{attribute 'object_name' := 'sta_EOFFBusy'}
METHOD sta_EOFFBusy : BOOL
                        // state implemetation
//--------------------------------------------------------------------------------------
// Entry action
	IF (me.StateMachine.intState<>me.StateMachine.intStateLastCycle) THEN
		me.StateMachine.intStateLastCycle := me.StateMachine.intState;
	END_IF

	
//--------------------------------------------------------------------------------------
// Cyclic action
	IF (me.StateMachine.intState=me.StateMachine.intStateLastCycle) THEN
		
		// In case of an emergency, set all childs to off 
		// Set in cyclic action because of possible errors or manual/auto changes!
		SUPER^.SetAllChildCmd(BASE_PLC.cCMD_OFF);

		// check if all childs have reached the state
		IF CheckAllChildState(cSTA_OFF) THEN
			me.StateMachine.intStateNext := cSTA_EOFF;
		END_IF
	END_IF

	
//--------------------------------------------------------------------------------------
// Exit action
	IF (me.StateMachine.intState<>me.StateMachine.intStateNext) THEN
		;
	END_IF
                      
END_METHOD

{attribute 'object_name' := 'sta_STOP'}
METHOD sta_STOP : BOOL
                        // state implemetation
//--------------------------------------------------------------------------------------
// Entry action
	IF (me.StateMachine.intState<>me.StateMachine.intStateLastCycle) THEN
		me.StateMachine.intStateLastCycle := me.StateMachine.intState;
	END_IF


//--------------------------------------------------------------------------------------
// Cyclic action
	IF (me.StateMachine.intState=me.StateMachine.intStateLastCycle) THEN
		
		// State Change Condition
		IF (me.Alarm.eActivAlmClass<E_AlmClass.TSTOP) THEN
			IF (me.intCmd=cCMD_RUN) THEN
				IF (SIf_In^.bolReady.intern OR SIf_Cfg^.bolIgnoreReadyInput) THEN 
					me.StateMachine.intStateNext := cSTA_RUNBusy;
				ELSE
					//SIf_MOD.Alm[E_ALM_MOD.NextModuleNotReadyWarning].strText := 'Next Module is not Ready';
					pfbAlarmCtrl^.setAlarm(CIf.Info.intCtrlId,E_ALM_MOD.NextModuleNotReadyWarning,0,ADR(SIf_MOD.Alm),E_AlmState.RST,CIf.Job.eMe_ActivAlmClass);
					CIf.Job.intACmd := cCMD_DONE;
				END_IF
			ELSIF (me.intCmd=cCMD_STANDBY) THEN
				IF (SIf_In^.bolReady.intern OR SIf_Cfg^.bolIgnoreReadyInput) THEN 
					me.StateMachine.intStateNext := cSTA_STANDBYBusy;
				ELSE
					//SIf_MOD.Alm[E_ALM_MOD.NextModuleNotReadyWarning].strText := 'Next Module is not Ready';
					pfbAlarmCtrl^.setAlarm(CIf.Info.intCtrlId,E_ALM_MOD.NextModuleNotReadyWarning,0,ADR(SIf_MOD.Alm),E_AlmState.RST,CIf.Job.eMe_ActivAlmClass);
					CIf.Job.intACmd := cCMD_DONE;
				END_IF
			END_IF
		END_IF
		
	END_IF

	
//--------------------------------------------------------------------------------------
// Exit action
	IF (me.StateMachine.intState<>me.StateMachine.intStateNext) THEN
		;
	END_IF
                      
END_METHOD

{attribute 'object_name' := 'sta_RUNBusy'}
METHOD sta_RUNBusy : BOOL
  VAR
    ii : INT;
    bolFurtherGrpExist : BOOL;
  END_VAR
                        // state implemetation
//--------------------------------------------------------------------------------------
// Entry action
	IF (me.StateMachine.intState<>me.StateMachine.intStateLastCycle) THEN
		me.StateMachine.intStateLastCycle := me.StateMachine.intState;
		// Init sub state machine
		me.SubStateMachine.intState := cSTA_SUB_INITIALIZED; 
		me.SubStateMachine.intStateNext := cSTA_SUB_INITIALIZED;
	END_IF

//--------------------------------------------------------------------------------------
// Cyclic action
	IF (me.StateMachine.intState=me.StateMachine.intStateLastCycle) THEN

		// Simulation
		IF (CIf.SwCfg.bolSimulation) THEN
			;
		END_IF
	
		// Start Cycle with substates	
		//--------------------------------------------------------------------------------------
		// sub state machine for sequence
		CASE me.SubStateMachine.intState OF
			//--------------------------------------------------------------------------------------
			cSTA_SUB_INITIALIZED:
			
				// Loop over all registered childs
				FOR ii:=0 TO usiNumOfSeq-1 BY 1 DO
					// Clear checked flag		
					aListOfSeq[ii].bolChecked:= FALSE;
				END_FOR
				uinGroupIndex:= 1;
				me.SubStateMachine.intStateNext := cSTA_SUB_SEND_GROUP_CMD;
				
			cSTA_SUB_SEND_GROUP_CMD:
				
				intCheckCounter:= 0;
				// Loop over all registered childs
				FOR ii:=0 TO usiNumOfSeq-1 BY 1 DO
					// If child is associated for the current group index		
					IF (aListOfSeq[ii].uinGroupRun = uinGroupIndex) THEN
						// Send defined command
						aListOfSeq[ii].pCIF^.Job.intACmd:= aListOfSeq[ii].intCmdSeqRun;
						intCheckCounter:= intCheckCounter + 1;
					END_IF			
				END_FOR
				// Change state
				me.SubStateMachine.intStateNext := cSTA_SUB_CHECK_GROUP_STATUS;
			
			
			cSTA_SUB_CHECK_GROUP_STATUS:
	
				// Loop over all registered childs
				FOR ii:=0 TO usiNumOfSeq-1 BY 1 DO
					// If child is associated for the current group index		
					IF (aListOfSeq[ii].uinGroupRun = uinGroupIndex) THEN
						// Check defined status and if child not already checked
						IF (((aListOfSeq[ii].pCIF^.Job.intState = aListOfSeq[ii].intStatusSeqRun) OR 
						(aListOfSeq[ii].pCIF^.Job.intState = aListOfSeq[ii].intStatusSeqRun2)) AND (aListOfSeq[ii].bolChecked = FALSE)) THEN
							aListOfSeq[ii].bolChecked:= TRUE;
							intCheckCounter:= intCheckCounter - 1;
						END_IF				
					END_IF			
				END_FOR
				
				// All childs in group has the right state
				IF (intCheckCounter <= 0) THEN		
					bolFurtherGrpExist:= FALSE;
					// Check if a further group exist!	
					FOR ii:=0 TO usiNumOfSeq-1 BY 1 DO	
						IF (aListOfSeq[ii].uinGroupRun > uinGroupIndex) THEN
							bolFurtherGrpExist:= TRUE;
							EXIT;
						END_IF			
					END_FOR
					// further group exist
					IF (bolFurtherGrpExist = TRUE) THEN
						IF (uinGroupIndex < uinMaxNrOfGroups) THEN			
							me.SubStateMachine.intStateNext := cSTA_SUB_WAIT;	
						END_IF
					ELSE
						me.SubStateMachine.intStateNext := cSTA_SUB_FINISHED;		
					END_IF
				END_IF

			cSTA_SUB_WAIT:
				
				IF (me.SubStateMachine.udiTimeInState_ms >= SIf_Par^.aListOfRunGrpWaitTime_ms[uinGroupIndex-1]) THEN
					// Inc. group index 
					uinGroupIndex:= uinGroupIndex + 1;	
					// Change state, send command for next group
					me.SubStateMachine.intStateNext := cSTA_SUB_SEND_GROUP_CMD;
				END_IF
			
			cSTA_SUB_FINISHED:
					;		
		END_CASE
		
		// Check time out error
		IF (SIf_MOD.Par^.udiTimeoutStarting_ms <> 0) AND (me.SubStateMachine.udiTimeInState_ms > (SIf_Par^.aListOfRunGrpWaitTime_ms[uinGroupIndex-1] + SIf_MOD.Par^.udiTimeoutStarting_ms)) THEN
			//SIf_MOD.Alm[E_ALM_MOD.TimeoutStarGroup].strText := 'Timeout start group';
			pfbAlarmCtrl^.setAlarm(CIf.Info.intCtrlId,E_ALM_MOD.TimeoutStartGroup,uinGroupIndex,ADR(SIf_MOD.Alm),E_AlmState.RST,CIf.Job.eMe_ActivAlmClass);
			me.StateMachine.intStateNext := cSTA_ERROR;
		END_IF
		
		// State Change Condition
		IF (me.intCmd=cCMD_STOP) THEN
			me.StateMachine.intStateNext :=  cSTA_STOPBusy;
		ELSIF NOT (SIf_In^.bolReady.intern OR SIf_Cfg^.bolIgnoreReadyInput) THEN
			//SIf_MOD.Alm[E_ALM_MOD.NextModuleNotReadyStop].strText := 'Next Module is not Ready';
			pfbAlarmCtrl^.setAlarm(CIf.Info.intCtrlId,E_ALM_MOD.NextModuleNotReadyStop,0,ADR(SIf_MOD.Alm),E_AlmState.RST,CIf.Job.eMe_ActivAlmClass);
			me.StateMachine.intStateNext := cSTA_STOPBusy;
			CIf.Job.intACmd := cCMD_DONE;
		ELSIF (me.SubStateMachine.intState = cSTA_SUB_FINISHED) THEN
			me.StateMachine.intStateNext := cSTA_RUN;
		END_IF
	END_IF

//--------------------------------------------------------------------------------------
// Exit action
	IF (me.StateMachine.intState<>me.StateMachine.intStateNext) THEN
		;
	END_IF
                      
END_METHOD

{attribute 'object_name' := 'CheckAllChildStateOr'}
METHOD CheckAllChildStateOr : BOOL
  VAR_INPUT
    In_intCheckState1 : INT;
    In_intCheckState2 : INT;
  END_VAR
  VAR
    uinIdx : UINT;
  END_VAR
                        // check if all child controller have reached one of the two In_intCheckState
CheckAllChildStateOr := TRUE;
IF (CIf.Info.uinChildNbr > 0) THEN
	FOR uinIdx := 0 TO CIf.Info.uinChildNbr - 1 DO
		CheckAllChildStateOr := CheckAllChildStateOr AND ((CIf.Info.p_aCIf[uinIdx]^.Job.intState = In_intCheckState1) OR (CIf.Info.p_aCIf[uinIdx]^.Job.intState = In_intCheckState2));
		IF (CheckAllChildStateOr=FALSE) THEN	// at least one child has not whished state reached
			EXIT ;
		END_IF 
	END_FOR
END_IF
                      
END_METHOD

{attribute 'object_name' := 'CtrlInit'}
METHOD CtrlInit : BOOL
  VAR
    ii : INT;
  END_VAR
                        SUPER^.CtrlInit();

// Initialize all child controller
// Childs are listed in list of sequences
FOR ii:=0 TO usiNumOfSeq-1 BY 1 DO	
	aListOfSeq[ii].pCIF := THIS^.AddChild(aListOfSeq[ii].pChild^);
END_FOR

_fbSignalTower.Initialize();
_fbSignalTower.HornEnable := SIf_MOD.Cfg^.bolStackLightHornEnable;

                      
END_METHOD

{attribute 'object_name' := 'sta_EOFF'}
METHOD sta_EOFF : BOOL
                        // state implemetation
//--------------------------------------------------------------------------------------
// Entry action
	IF (me.StateMachine.intState<>me.StateMachine.intStateLastCycle) THEN
		me.StateMachine.intStateLastCycle := me.StateMachine.intState;	
	END_IF

//--------------------------------------------------------------------------------------
// Cyclic action
	IF (me.StateMachine.intState=me.StateMachine.intStateLastCycle) THEN		
		
		// As long as the EMO is not reseted!
		IF NOT (SIf_In^.bolEmoOk.intern) THEN
			// Clear pending and new commands cyclic to prevent automatic recovery!
			CIf.Job.intACmd := BASE_PLC.cCMD_DONE;
			CIf.Job.intMCmd := BASE_PLC.cCMD_DONE;
		END_IF
	
		// State Change Condition
		IF (SIf_In^.bolEmoOk.intern) AND (me.Alarm.eActivAlmClass<>E_AlmClass.EOFF) AND (me.intCmd<>BASE_PLC.cCMD_EOFF) AND (me.intCmd<>BASE_PLC.cCMD_DONE) THEN
			me.StateMachine.intStateNext := cSTA_OFF;
		END_IF
	END_IF

//--------------------------------------------------------------------------------------
// Exit action
	IF (me.StateMachine.intState<>me.StateMachine.intStateNext) THEN
		;
	END_IF
                      
END_METHOD

{attribute 'object_name' := 'checkValidPointer'}
METHOD checkValidPointer : BOOL
                        IF (usiNumOfSeq = usiNumOfValidPointerSeqChild) AND (SIf_Cfg<>0) AND (SIf_Par<>0) AND (SIf_Cur<>0) AND (SIf_In<>0) THEN
	checkValidPointer:= TRUE;
ELSE
	// Invalid child pointer
	checkValidPointer:= FALSE;	
	//SIf_MOD.Alm[E_ALM_MOD.InvalidPointer].strText := 'Invalid pointer';
	pfbAlarmCtrl^.setAlarm(CIf.Info.intCtrlId,E_ALM_MOD.InvalidPointer,0,ADR(SIf_MOD.Alm),E_AlmState.RST,CIf.Job.eMe_ActivAlmClass);	
END_IF
                      
END_METHOD

{attribute 'object_name' := 'AddIBufferFullChilds'}
METHOD AddIBufferFullChilds
  VAR_INPUT
    pFB_ChildTypeIBuffer : POINTER TO FB_IBuffer;
  END_VAR
                        // Method add childs with BufferFull information to the array
IF (usiNumOfIBufferFullChild <= (Base_Const.cMaxNrOfChilds-1)) THEN
	// Add child controller to list
	a_IBufferFullChildCtrl[usiNumOfIBufferFullChild] := pFB_ChildTypeIBuffer^;

	// Inc. number of IBufferFull childs
	usiNumOfIBufferFullChild:= usiNumOfIBufferFullChild+1;
END_IF


                      
END_METHOD

{attribute 'object_name' := 'sta_STANDBY'}
METHOD sta_STANDBY : BOOL
                        // state implemetation
//--------------------------------------------------------------------------------------
// Entry action
	IF (me.StateMachine.intState<>me.StateMachine.intStateLastCycle) THEN
		me.StateMachine.intStateLastCycle := me.StateMachine.intState;
	END_IF


//--------------------------------------------------------------------------------------
// Cyclic action
	IF (me.StateMachine.intState=me.StateMachine.intStateLastCycle) THEN
		
		// State Change Condition
		IF (me.Alarm.eActivAlmClass<E_AlmClass.TSTOP) THEN
			IF (me.intCmd=cCMD_RUN) THEN
				IF (SIf_In^.bolReady.intern OR SIf_Cfg^.bolIgnoreReadyInput) THEN 
					me.StateMachine.intStateNext := cSTA_RUNBusy;
				ELSE
					//SIf_MOD.Alm[E_ALM_MOD.NextModuleNotReadyWarning].strText := 'Next Module is not Ready';
					pfbAlarmCtrl^.setAlarm(CIf.Info.intCtrlId,E_ALM_MOD.NextModuleNotReadyWarning,0,ADR(SIf_MOD.Alm),E_AlmState.RST,CIf.Job.eMe_ActivAlmClass);
					CIf.Job.intACmd := cCMD_DONE;
				END_IF
			END_IF
			
			IF (me.intCmd=cCMD_STOP) THEN
					me.StateMachine.intStateNext := cSTA_STOPBusy;
			END_IF
		END_IF
	END_IF

//--------------------------------------------------------------------------------------
// Exit action
	IF (me.StateMachine.intState<>me.StateMachine.intStateNext) THEN
		;
	END_IF
                      
END_METHOD

{attribute 'object_name' := 'CycleEndDuty'}
METHOD CycleEndDuty : BOOL
                        CycleEndDuty := SUPER^.CycleEndDuty();

_fbSignalTower.State := me.StateMachine.intState;
_fbSignalTower.AlarmClass := me.Alarm.eActivAlmClass;
_fbSignalTower();
Out_bolRed 		:= _fbSignalTower.Out_bolRed;
Out_bolYellow 	:= _fbSignalTower.Out_bolYellow;
Out_bolGreen 	:= _fbSignalTower.Out_bolGreen;
Out_bolBlue 	:= _fbSignalTower.Out_bolBlue;
Out_bolHorn 	:= _fbSignalTower.Out_bolHorn;

                      
END_METHOD

{attribute 'object_name' := 'IoInBridge'}
METHOD IoInBridge : BOOL
                        // digitale and analoge inputs read from hardware or forcing
SIf_In^.bolReady.map	:= THIS^.In_bolReady;
SIf_In^.bolEmoOk.map	:= THIS^.In_bolEmoOk;

IF (CIf.SwCfg.bolSimulation = FALSE) THEN
	BASE_PLC.getInBol(CIf.Job.bolIoForce,ADR(SIf_In^.bolReady));
	BASE_PLC.getInBol(CIf.Job.bolIoForce,ADR(SIf_In^.bolEmoOk));
ELSE
	//simulation of global IO
	SIf_In^.bolReady.intern	:= TRUE;
	SIf_In^.bolEmoOk.intern	:= TRUE;
END_IF
                      
END_METHOD

{attribute 'object_name' := 'AddSeqChild'}
METHOD AddSeqChild
  VAR_INPUT
    stSequence : T_Sequence;
  END_VAR
                        // Method add a sequence to list
IF (usiNumOfSeq <= (Base_Const.cMaxNrOfChilds-1)) THEN
	aListOfSeq[usiNumOfSeq].pChild:= stSequence.pChild;
	aListOfSeq[usiNumOfSeq].uinGroupRun:= stSequence.uinGroupRun;
	aListOfSeq[usiNumOfSeq].uinGroupStop:= stSequence.uinGroupStop;
	aListOfSeq[usiNumOfSeq].intCmdSeqRun:= stSequence.intCmdSeqRun;
	aListOfSeq[usiNumOfSeq].intStatusSeqRun:= stSequence.intStatusSeqRun;
	aListOfSeq[usiNumOfSeq].intStatusSeqRun2:= stSequence.intStatusSeqRun2;
	aListOfSeq[usiNumOfSeq].intCmdSeqStop:= stSequence.intCmdSeqStop;
	aListOfSeq[usiNumOfSeq].intStatusSeqStop:= stSequence.intStatusSeqStop;	
	aListOfSeq[usiNumOfSeq].intStatusSeqStop2:= stSequence.intStatusSeqStop2;
	aListOfSeq[usiNumOfSeq].intCmdSeqStandby:= stSequence.intCmdSeqStandby;
	aListOfSeq[usiNumOfSeq].intStatusSeqStandby:= stSequence.intStatusSeqStandby;
	aListOfSeq[usiNumOfSeq].intStatusSeqStandby2:= stSequence.intStatusSeqStandby2;
	// Inc. number of sequence
	usiNumOfSeq:= usiNumOfSeq+1;
	// Check if the pointer is valid
	IF (stSequence.pChild<>0) THEN
		usiNumOfValidPointerSeqChild:= usiNumOfValidPointerSeqChild+1;
	END_IF
END_IF
                      
END_METHOD

{attribute 'object_name' := 'sta_PONBusy'}
METHOD sta_PONBusy : BOOL
                        // state implemetation
//--------------------------------------------------------------------------------------
// Entry action
	IF (me.StateMachine.intState<>me.StateMachine.intStateLastCycle) THEN
		me.StateMachine.intStateLastCycle := me.StateMachine.intState;
		
		SetAllChildCmd(cCMD_PON); // set acmd off all childs 
	END_IF


//--------------------------------------------------------------------------------------
// Cyclic action
	IF (me.StateMachine.intState=me.StateMachine.intStateLastCycle) THEN

		// State Change Condition
		IF (FALSE) THEN
			;
		ELSIF CheckAllChildStateOr(cSTA_PON, cSTA_RUN) THEN
			me.StateMachine.intStateNext := cSTA_PON;
		END_IF
		
	END_IF


//--------------------------------------------------------------------------------------
// Exit action
	IF (me.StateMachine.intState<>me.StateMachine.intStateNext) THEN
		;
	END_IF
                      
END_METHOD

{attribute 'object_name' := 'sta_STOPBusy'}
METHOD sta_STOPBusy : BOOL
  VAR
    ii : INT;
    bolFurtherGrpExist : BOOL;
  END_VAR
                        // state implemetation
//--------------------------------------------------------------------------------------
// Entry action
	IF (me.StateMachine.intState<>me.StateMachine.intStateLastCycle) THEN
		me.StateMachine.intStateLastCycle := me.StateMachine.intState;	
		// Init sub state machine
		me.SubStateMachine.intState := cSTA_SUB_INITIALIZED; 
		me.SubStateMachine.intStateNext := cSTA_SUB_INITIALIZED;
	END_IF


//--------------------------------------------------------------------------------------
// Cyclic action
	IF (me.StateMachine.intState=me.StateMachine.intStateLastCycle) THEN

		// Simulation
		IF (CIf.SwCfg.bolSimulation) THEN
			;
		END_IF
		
		// Stop Cycle with substates	
		//--------------------------------------------------------------------------------------
		// sub state machine for sequence
		CASE me.SubStateMachine.intState OF
			//--------------------------------------------------------------------------------------
			cSTA_SUB_INITIALIZED:
			
				// Loop over all registered childs
				FOR ii:=0 TO usiNumOfSeq-1 BY 1 DO
					// Clear checked flag		
					aListOfSeq[ii].bolChecked:= FALSE;
				END_FOR
				uinGroupIndex:= 1;
				me.SubStateMachine.intStateNext := cSTA_SUB_SEND_GROUP_CMD;
				
			cSTA_SUB_SEND_GROUP_CMD:
				
				intCheckCounter:= 0;
				// Loop over all registered childs
				FOR ii:=0 TO usiNumOfSeq-1 BY 1 DO
					// If child is associated for the current group index		
					IF (aListOfSeq[ii].uinGroupStop = uinGroupIndex) THEN
						// Send defined command
						aListOfSeq[ii].pCIF^.Job.intACmd:= aListOfSeq[ii].intCmdSeqStop;
						intCheckCounter:= intCheckCounter + 1;
					END_IF			
				END_FOR
				// Change state
				me.SubStateMachine.intStateNext := cSTA_SUB_CHECK_GROUP_STATUS;
			
			
			cSTA_SUB_CHECK_GROUP_STATUS:
	
				// Loop over all registered childs
				FOR ii:=0 TO usiNumOfSeq-1 BY 1 DO
					// If child is associated for the current group index		
					IF (aListOfSeq[ii].uinGroupStop = uinGroupIndex) THEN
						// Check defined status and if child not already checked
						IF (((aListOfSeq[ii].pCIF^.Job.intState = aListOfSeq[ii].intStatusSeqStop) OR (aListOfSeq[ii].pCIF^.Job.intState = aListOfSeq[ii].intStatusSeqStop2)) AND (aListOfSeq[ii].bolChecked = FALSE)) THEN
							aListOfSeq[ii].bolChecked:= TRUE;
							intCheckCounter:= intCheckCounter - 1;
						END_IF				
					END_IF			
				END_FOR
				
				// All childs in group has the right state
				IF (intCheckCounter <= 0) THEN		
					bolFurtherGrpExist:= FALSE;
					// Check if a further group exist!	
					FOR ii:=0 TO usiNumOfSeq-1 BY 1 DO	
						IF (aListOfSeq[ii].uinGroupStop > uinGroupIndex) THEN
							bolFurtherGrpExist:= TRUE;
							EXIT;
						END_IF			
					END_FOR
					// further group exist
					IF (bolFurtherGrpExist = TRUE) THEN
						IF (uinGroupIndex < uinMaxNrOfGroups) THEN			
							me.SubStateMachine.intStateNext := cSTA_SUB_WAIT;	
						END_IF
					ELSE
						me.SubStateMachine.intStateNext := cSTA_SUB_FINISHED;		
					END_IF
				END_IF

			cSTA_SUB_WAIT:
				
				IF (me.SubStateMachine.udiTimeInState_ms >= SIf_Par^.aListOfStopGrpWaitTime_ms[uinGroupIndex-1]) THEN
					// Inc. group index 
					uinGroupIndex:= uinGroupIndex + 1;	
					// Change state, send command for next group
					me.SubStateMachine.intStateNext := cSTA_SUB_SEND_GROUP_CMD;
				END_IF
			
			cSTA_SUB_FINISHED:
					;		
		END_CASE
		
		// Check time out error
		IF (SIf_MOD.Par^.udiTimeoutStopping_ms <> 0) AND (me.SubStateMachine.udiTimeInState_ms > (SIf_Par^.aListOfStopGrpWaitTime_ms[uinGroupIndex-1] + SIf_MOD.Par^.udiTimeoutStopping_ms)) THEN
			//SIf_MOD.Alm[E_ALM_MOD.TimeoutStopGroup].strText := 'Timeout stop group';
			pfbAlarmCtrl^.setAlarm(CIf.Info.intCtrlId,E_ALM_MOD.TimeoutStopGroup,uinGroupIndex,ADR(SIf_MOD.Alm),E_AlmState.RST,CIf.Job.eMe_ActivAlmClass);
			me.StateMachine.intStateNext := cSTA_ERROR;
		END_IF
	
		// State Change Condition
		IF (me.SubStateMachine.intState = cSTA_SUB_FINISHED) THEN
			me.StateMachine.intStateNext := cSTA_STOP;
		ELSIF (me.intCmd=cCMD_RUN) THEN
			// State Change Condition
			IF (me.Alarm.eActivAlmClass<E_AlmClass.TSTOP) THEN	
				me.StateMachine.intStateNext := cSTA_RUNBusy;	
			ELSE
				// Clear pending command to prevent automatic recovery!
				CIf.Job.intACmd:=cSTA_DONE;
			END_IF
		END_IF

	END_IF

//--------------------------------------------------------------------------------------
// Exit action
	IF (me.StateMachine.intState<>me.StateMachine.intStateNext) THEN
		;
	END_IF
                      
END_METHOD

{attribute 'object_name' := 'sta_OFFBusy'}
METHOD sta_OFFBusy : BOOL
                        // state implemetation
//--------------------------------------------------------------------------------------
// Entry action
	IF (me.StateMachine.intState<>me.StateMachine.intStateLastCycle) THEN
		me.StateMachine.intStateLastCycle := me.StateMachine.intState;
		
		// Set commandos not only in entry action because of possible errors or manual/auto changes
		// PRE/AVME 06.01.2014
		//SetAllChildCmd(cCMD_OFF); // set acmd off all childs 
	END_IF


//--------------------------------------------------------------------------------------
// Cyclic action
	IF (me.StateMachine.intState=me.StateMachine.intStateLastCycle) THEN
		
		SetAllChildCmd(cCMD_OFF); // set acmd off all childs 
		
		// State Change Condition
		IF (CheckAllChildState(cSTA_OFF)) THEN
			me.StateMachine.intStateNext := cSTA_OFF;
		ELSIF (me.intCmd=cCMD_RUN) AND (me.Alarm.eActivAlmClass < E_AlmClass.TSTOP) THEN
			me.StateMachine.intStateNext := cSTA_RUNBusy;
		END_IF
	END_IF


//--------------------------------------------------------------------------------------
// Exit action
	IF (me.StateMachine.intState<>me.StateMachine.intStateNext) THEN
		;
	END_IF
                      
END_METHOD

{attribute 'object_name' := 'FB_init'}
METHOD FB_init : BOOL
  VAR_INPUT
    bInitRetains : BOOL;  (* if TRUE, the retain variables are initialized (warm start / cold start) *)
    bInCopyCode : BOOL;  (* if TRUE, the instance afterwards gets moved into the copy code (online change) *)
  END_VAR
  VAR
    ii : UINT;
  END_VAR
                        // to manually change in new FUB implementation!!!
// define valid commands for this controller
FOR ii:= 0 TO (SIZEOF(CIf.Job.aCmdList)/SIZEOF(CIf.Job.aCmdList[0])-1) BY 1 DO
	IF (CIf.Job.aCmdList[ii].intCmd=cCMD_INITIALIZED) THEN
		// found first empty array element
		EXIT;
	END_IF
END_FOR

CIf.Job.aCmdList[ii].intCmd := cCMD_RUN;
CIf.Job.aCmdList[ii].strName := 'Run'; 
CIf.Job.aCmdList[ii].bolAvailable := TRUE;
ii := ii +1;
CIf.Job.aCmdList[ii].intCmd := cCMD_STOP;
CIf.Job.aCmdList[ii].strName := 'Stop'; 
CIf.Job.aCmdList[ii].bolAvailable := TRUE;
ii := ii +1;
CIf.Job.aCmdList[ii].intCmd := cCMD_STANDBY;
CIf.Job.aCmdList[ii].strName := 'Standby'; 
CIf.Job.aCmdList[ii].bolAvailable := TRUE;
ii := ii +1;

// set name of class/typ
CIf.Info.strType := 'FB_CtrlModule';
CIf.Info.strFullName := 'Base Controller Module';

// set alarm class
SIf_MOD.Alm[E_ALM_MOD.InvalidPointer].eAlmClass := E_AlmClass.STOP;
SIf_MOD.Alm[E_ALM_MOD.InvalidPointer].strText := 'Invalid pointer';
SIf_MOD.Alm[E_ALM_MOD.CommunicationError].eAlmClass := E_AlmClass.OFF;
SIf_MOD.Alm[E_ALM_MOD.CommunicationError].strText := 'Communication error to line control';
SIf_MOD.Alm[E_ALM_MOD.EmergencyOff].eAlmClass := E_AlmClass.EOFF;
SIf_MOD.Alm[E_ALM_MOD.EmergencyOff].strText := 'Emergency off active';
SIf_MOD.Alm[E_ALM_MOD.TimeoutStartGroup].eAlmClass := E_AlmClass.OFF;
SIf_MOD.Alm[E_ALM_MOD.TimeoutStartGroup].strText := 'Timeout start group';
SIf_MOD.Alm[E_ALM_MOD.TimeoutStopGroup].eAlmClass := E_AlmClass.OFF;
SIf_MOD.Alm[E_ALM_MOD.TimeoutStopGroup].strText := 'Timeout stop group';
SIf_MOD.Alm[E_ALM_MOD.NextModuleNotReadyWarning].eAlmClass := E_AlmClass.WARNING;
SIf_MOD.Alm[E_ALM_MOD.NextModuleNotReadyWarning].strText := 'Next Module is not Ready';
SIf_MOD.Alm[E_ALM_MOD.NextModuleNotReadyStop].eAlmClass := E_AlmClass.STOP;
SIf_MOD.Alm[E_ALM_MOD.NextModuleNotReadyStop].strText := 'Next Module is not Ready';

//*******************************************************************************
// initial values
//*******************************************************************************
udinTimeToggle_ms := 0;
// software configuration
CIf.SwCfg.bolExist := TRUE;
CIf.SwCfg.bolSimulation := FALSE;

me.AlarmConfig.bolChildrenAlarmPropagation := FALSE;

// No initialization for cfg and par in this base module!
// Pointer address of the property is not defined at this time
                      
END_METHOD

{attribute 'object_name' := 'AddIBufferChilds'}
METHOD AddIBufferChilds
  VAR_INPUT
    pFB_ChildTypeIBuffer : POINTER TO FB_IBuffer;
  END_VAR
                        // Method add childs with type of IBuffer to the array
IF (usiNumOfIBufferChild <= (Base_Const.cMaxNrOfChilds-1)) THEN
	// Add child controller to list
	a_IBufferChildCtrl[usiNumOfIBufferChild] := pFB_ChildTypeIBuffer^;
	// Inc. number of IBuffer childs
	usiNumOfIBufferChild:= usiNumOfIBufferChild+1;
END_IF


                      
END_METHOD

{attribute 'object_name' := 'StateMachine'}
METHOD StateMachine : BOOL
                        SUPER^.StateMachine();

// main statemachine of base controller
CASE me.StateMachine.intState OF
	cSTA_RUN: 
        THIS^.sta_RUN();
    cSTA_RUNBusy: 
        THIS^.sta_RUNBusy();
	cSTA_STOP: 
        THIS^.sta_STOP();
    cSTA_STOPBusy: 
        THIS^.sta_STOPBusy();
	cSTA_STANDBY:
		THIS^.sta_STANDBY();
	cSTA_STANDBYBusy:
		THIS^.sta_STANDBYBusy();
END_CASE;
                      
END_METHOD

{attribute 'object_name' := 'checkChildAlmClass'}
METHOD checkChildAlmClass : BOOL
                        //------------------------------------------------------------------------------------------------------
// check child alarm classes
// set me alarm class active if at least one child has an EOFF
IF CheckAllChildAlmClass(E_AlmClass.EOFF) THEN
	CIf.Job.eMe_ActivAlmClass := E_AlmClass.EOFF;
	me.Alarm.bolfp := TRUE;
ELSIF CheckAllChildAlmClass(E_AlmClass.OFF) THEN
	CIf.Job.eMe_ActivAlmClass := E_AlmClass.OFF;
	me.Alarm.bolfp := TRUE;
ELSIF CheckAllChildAlmClass(E_AlmClass.STOP) THEN
	CIf.Job.eMe_ActivAlmClass := E_AlmClass.STOP;
	me.Alarm.bolfp := TRUE;
ELSIF CheckAllChildAlmClass(E_AlmClass.TSTOP) THEN
	CIf.Job.eMe_ActivAlmClass := E_AlmClass.TSTOP;
	me.Alarm.bolfp := TRUE;
ELSE
	IF (me.Alarm.bolfp) THEN
		CIf.Job.eMe_ActivAlmClass := E_AlmClass.NONE; // no reset necessary
		me.Alarm.bolfp := FALSE;
	END_IF
END_IF

//------------------------------------------------------------------------------------------------------
// set alarm class parent of childs
//------------------------------------------------------------------------------------------------------
// set alarm class parent of childs in the case of a parent EOFF or me=OFF or EOFF
IF (CIf.Job.eParent_ActivAlmClass=E_AlmClass.EOFF) THEN
	SetAllChildAlmClass(CIf.Job.eParent_ActivAlmClass);
ELSIF(CIf.Job.eMe_ActivAlmClass=E_AlmClass.EOFF) OR (CIf.Job.eMe_ActivAlmClass=E_AlmClass.OFF) THEN
	SetAllChildAlmClass(CIf.Job.eMe_ActivAlmClass);
ELSE
	// no important alarm for child active
	SetAllChildAlmClass(E_AlmClass.NONE);
END_IF
                      
END_METHOD

{attribute 'object_name' := 'FurtherReactions'}
METHOD FurtherReactions : BOOL
                        IF		(me.Alarm.eActivAlmClass=E_AlmClass.STOP)
	AND (me.StateMachine.intState<>cSTA_ERROR)		AND	(me.StateMachine.intState<>cSTA_ERRORQuit)
	AND	(me.StateMachine.intState<>cSTA_EOFF)		AND	(me.StateMachine.intState<>cSTA_EOFFBusy)
	AND	(me.StateMachine.intState<>cSTA_OFF)		AND	(me.StateMachine.intState<>cSTA_OFFBusy)
	AND (me.StateMachine.intState<>cSTA_STOP)		AND (me.StateMachine.intState<>cSTA_STOPBusy)
	AND	(me.StateMachine.intState>cSTA_PON) THEN
	
	me.StateMachine.intStateNext := cSTA_STOPBusy;
	CIf.Job.intACmd := cCMD_DONE;
	CIf.Job.intMCmd := cCMD_DONE;
	
ELSIF	(me.Alarm.eActivAlmClass=E_AlmClass.TSTOP)
	AND (me.StateMachine.intState<>cSTA_ERROR)		AND	(me.StateMachine.intState<>cSTA_ERRORQuit)
	AND	(me.StateMachine.intState<>cSTA_EOFF)		AND	(me.StateMachine.intState<>cSTA_EOFFBusy)
	AND	(me.StateMachine.intState<>cSTA_OFF)		AND	(me.StateMachine.intState<>cSTA_OFFBusy)
	AND (me.StateMachine.intState<>cSTA_STOP)		AND (me.StateMachine.intState<>cSTA_STOPBusy)
	AND	(me.StateMachine.intState>cSTA_PON) THEN
	
	me.StateMachine.intStateNext := cSTA_STOPBusy;
	CIf.Job.intACmd := cCMD_DONE;
	CIf.Job.intMCmd := cCMD_DONE;
	
END_IF
                      
END_METHOD

{attribute 'object_name' := 'sta_ERROR'}
METHOD sta_ERROR : BOOL
                        // state implemetation
//--------------------------------------------------------------------------------------
// Entry action
	IF (me.StateMachine.intState<>me.StateMachine.intStateLastCycle) THEN
		me.StateMachine.intStateHistory := me.StateMachine.intStateLastCycle; // -> possibillity to go back to state before error
		me.StateMachine.intStateLastCycle := me.StateMachine.intState;
		// Clear pending command to prevent automatic recovery!
		CIf.Job.intACmd:=cSTA_DONE;
		// In case on an error, set all childs to off
		SetAllChildCmd(cCMD_OFF);
	END_IF

//--------------------------------------------------------------------------------------
// Cyclic action
	IF (me.StateMachine.intState=me.StateMachine.intStateLastCycle) THEN
		
		;
		// State Change Condition
		IF ((CIf.Job.bolAlmReset = TRUE) AND (CheckAllChildState(cSTA_OFF))) THEN
			me.StateMachine.intStateNext := cSTA_ERRORQuit;
		END_IF
	END_IF

//--------------------------------------------------------------------------------------
// Exit action
	IF (me.StateMachine.intState<>me.StateMachine.intStateNext) THEN
		;
	END_IF
                      
END_METHOD

PROPERTY SIf_Out : POINTER TO T_Ctrl_SIf_MOD_Out
GET
                          SIf_Out:= SIf_MOD.Out; 
                        
END_GET
SET
                          SIf_MOD.Out := SIf_Out;
                        
END_SET
END_PROPERTY

PROPERTY SIf_Cur : POINTER TO T_Ctrl_SIf_MOD_Cur
GET
                          SIf_Cur:= SIf_MOD.Cur; 
                        
END_GET
SET
                          SIf_MOD.Cur := SIf_Cur; 
                        
END_SET
END_PROPERTY

PROPERTY SIf_Par : POINTER TO T_Ctrl_SIf_MOD_Par
GET
                          SIf_Par:= SIf_MOD.Par; 
                        
END_GET
SET
                          SIf_MOD.Par := SIf_Par; 
                        
END_SET
END_PROPERTY

PROPERTY SIf_In : POINTER TO T_Ctrl_SIf_MOD_In
GET
                          SIf_In:= SIf_MOD.In; 
                        
END_GET
SET
                          SIf_MOD.In := SIf_In;
                        
END_SET
END_PROPERTY

PROPERTY SIf_Cfg : POINTER TO T_Ctrl_SIf_MOD_Cfg
GET
                          SIf_Cfg:= SIf_MOD.Cfg; 
                        
END_GET
SET
                          SIf_MOD.Cfg := SIf_Cfg;
                        
END_SET
END_PROPERTY
END_FUNCTION_BLOCK

(* FUNCTION_BLOCK PUBLIC FB_IBuffer IMPLEMENTS IBuffer *)
FUNCTION_BLOCK FB_IBuffer EXTENDS FB_CtrlBase IMPLEMENTS IBuffer

                  // This is a Dummy-FB, used for the interface (IBuffer) to the buffer-modules
                

PROPERTY NumOfItems : DINT
GET
                          
                        
END_GET
END_PROPERTY

PROPERTY MaxCapacity : DINT
GET
                          
                        
END_GET
END_PROPERTY

PROPERTY BufferFull : BOOL
GET
                          
                        
END_GET
END_PROPERTY
END_FUNCTION_BLOCK

FUNCTION_BLOCK FB_GHT IMPLEMENTS IGHT
  VAR CONSTANT
    MAX_HASH_LISTS : INT := 3;
    MAX_HASHLIST_ENTRIES : INT := 50;
    CUTOFF_A : ULINT := 4000000000;
    CUTOFF_B : ULINT := 8000000000;
  END_VAR
  VAR
    m_bolDeleteItems : BOOL;
    m_uintCount : UINT;
    m_fbHashTable : ARRAY[0..(MAX_HASH_LISTS - 1)] OF FB_HashTableCtrl;
    m_hHashTable : ARRAY[0..(MAX_HASH_LISTS - 1)] OF T_HHASHTABLE;
    m_uliCutoff : ARRAY[0..(MAX_HASH_LISTS - 1)] OF ULINT;
    m_aHashTableBuffer : ARRAY[0..(MAX_HASH_LISTS - 1)] OF T_GHTHashTableBuffer;
  END_VAR

                  
                

{attribute 'object_name' := 'Initialize'}
METHOD Initialize : BOOL
                        F_CreateHashTableHnd( ADR( m_aHashTableBuffer[0].aBuffer ), SIZEOF( m_aHashTableBuffer[0].aBuffer ), m_hHashTable[0] );
F_CreateHashTableHnd( ADR( m_aHashTableBuffer[1].aBuffer ), SIZEOF( m_aHashTableBuffer[1].aBuffer ), m_hHashTable[1] );
F_CreateHashTableHnd( ADR( m_aHashTableBuffer[2].aBuffer ), SIZEOF( m_aHashTableBuffer[2].aBuffer ), m_hHashTable[2] );
                      
END_METHOD

{attribute 'object_name' := 'GetTableIdx'}
METHOD GetTableIdx : INT
  VAR_INPUT
    uliBarcode : ULINT;
  END_VAR
                        IF uliBarcode < CUTOFF_A THEN
	GetTableIdx := 0;
	RETURN;
END_IF

IF uliBarcode > CUTOFF_B THEN
	GetTableIdx := 2;
	RETURN;
END_IF

GetTableIdx := 1;

                      
END_METHOD

{attribute 'object_name' := 'Lookup'}
METHOD Lookup : POINTER TO BYTE
  VAR_INPUT
    uliKey : ULINT;
    bolRemove : BOOL;
  END_VAR
  VAR
    pfbHashTable : POINTER TO FB_HashTableCtrl;
    phHashTable : POINTER TO T_HHASHTABLE;
    uliCutoff : ULINT;
    iIdx : INT;
  END_VAR
                        iIdx := GetTableIdx(uliKey);

m_fbHashTable[iIdx].A_Lookup( key := ULINT_TO_UDINT(uliKey-m_uliCutoff[iIdx]), hTable := m_hHashTable[iIdx] );

IF m_fbHashTable[iIdx].bOk THEN
	Lookup := m_fbHashTable[iIdx].getValue;
	
	IF bolRemove THEN
		m_fbHashTable[iIdx].A_Remove( key := ULINT_TO_UDINT(uliKey-m_uliCutoff[iIdx]), hTable := m_hHashTable[iIdx]);

		IF m_fbHashTable[iIdx].bOk THEN
			m_uintCount := m_uintCount - 1;
		END_IF
	END_IF
ELSE
	Lookup := NULL;
END_IF
                      
END_METHOD

{attribute 'object_name' := 'Clear'}
METHOD Clear : BOOL
  VAR_INPUT
    bolFreePointer : BOOL;
  END_VAR
  VAR
    iIdx : INT;
    pData : POINTER TO BYTE;
  END_VAR
                        FOR iIdx := 0 TO MAX_HASH_LISTS - 1 DO
	IF bolFreePointer THEN
		m_fbHashTable[iIdx].A_GetFirst(hTable := m_hHashTable[iIdx]);

		WHILE m_fbHashTable[iIdx].bOk DO
			pData := m_fbHashTable[iIdx].getValue;
			__DELETE(pData);
			m_fbHashTable[iIdx].A_GetNext(hTable := m_hHashTable[iIdx]);
		END_WHILE
		
	END_IF
	
	m_fbHashTable[iIdx].A_RemoveAll(hTable := m_hHashTable[iIdx]);
END_FOR

m_uintCount := 0;

                      
END_METHOD

{attribute 'object_name' := 'FB_init'}
METHOD FB_init : BOOL
  VAR_INPUT
    bInitRetains : BOOL;  (* if TRUE, the retain variables are initialized (warm start / cold start) *)
    bInCopyCode : BOOL;  (* if TRUE, the instance afterwards gets moved into the copy code (online change) *)
  END_VAR
                        m_uliCutoff[0] := 0;
m_uliCutoff[1] := CUTOFF_A;
m_uliCutoff[2] := CUTOFF_B;

m_uintCount := 0;
                      
END_METHOD

{attribute 'object_name' := 'AddItem'}
METHOD AddItem : BOOL
  VAR_INPUT
    uliKey : ULINT;
    pData : POINTER TO BYTE;
  END_VAR
  VAR
    iIdx : INT;
  END_VAR
                        iIdx := GetTableIdx(uliKey);

m_fbHashTable[iIdx].A_Add( key := ULINT_TO_UDINT(uliKey-m_uliCutoff[iIdx]), putValue := pData, hTable := m_hHashTable[iIdx] );

IF m_fbHashTable[iIdx].bOk THEN
	m_uintCount := m_uintCount + 1;
END_IF
                      
END_METHOD

PROPERTY Count : UINT
GET
                          
                        
END_GET
END_PROPERTY
END_FUNCTION_BLOCK

FUNCTION_BLOCK FB_IdBaseRecvDch EXTENDS FB_DataChannelRecvBase IMPLEMENTS I_DataChannelRecv
  VAR
    m_pInputData : POINTER TO T_IdBase_DCH;  (* Saber Inteface Variables ----------------------------------------------------------------- *)
  END_VAR

                  SUPER^();
                

{attribute 'object_name' := 'GetData'}
METHOD GetData : BOOL
  VAR_INPUT
    udiDataSize : UDINT;
    pData : POINTER TO BYTE;
  END_VAR
                        GetData := FALSE;

IF m_eState = E_SaberPlcDHCState.DataReady THEN
	IF (udiDataSize > 0 ) AND (pData <> TC3_MEMMAN.NULL) THEN
		TC2_SYSTEM.MEMCPY(destAddr := pData, srcAddr := m_pInputData, n := udiDataSize);
		m_eState := E_SaberPlcDHCState.Acknowledge;	
		GetData := TRUE;
	END_IF	
END_IF
                      
END_METHOD

{attribute 'object_name' := 'InitChannel'}
METHOD InitChannel : BOOL
  VAR_INPUT
    udiDataSize : UDINT;
    pInputData : POINTER TO BYTE;
  END_VAR
                        InitChannel := FALSE;

IF udiDataSize > 0 THEN
	IF pInputData <> TC3_MEMMAN.NULL THEN
		m_uinDataSize := udiDataSize;
		m_pInputData := pInputData;
		m_eState := E_SaberPlcDHCState.Init;
		InitChannel := TRUE;
	END_IF
END_IF

                      
END_METHOD
END_FUNCTION_BLOCK

FUNCTION_BLOCK FB_IdBaseSendDch EXTENDS FB_DataChannelSendBase IMPLEMENTS I_DataChannelSend
  VAR
    m_pOutputData : POINTER TO T_IdBase_DCH;  (* Saber Inteface Variables ----------------------------------------------------------------- *)
  END_VAR

                  SUPER^();
                

{attribute 'object_name' := 'SendData'}
METHOD SendData : BOOL
  VAR_INPUT
    udiDataSize : UDINT;
    pData : POINTER TO BYTE;
  END_VAR
                        SendData := FALSE;

IF m_eState = E_PlcSaberDHCState.WaitForJob THEN
	IF (udiDataSize > 0 ) AND (pData <> TC3_MEMMAN.NULL) THEN
		TC2_SYSTEM.MEMCPY(destAddr := m_pOutputData, srcAddr := pData, n := udiDataSize);
		m_eState := E_PlcSaberDHCState.SendData;	
		SendData := TRUE;
	END_IF	
END_IF
                      
END_METHOD

{attribute 'object_name' := 'InitChannel'}
METHOD InitChannel : BOOL
  VAR_INPUT
    udiDataSize : UDINT;
    pOutputData : POINTER TO BYTE;
  END_VAR
                        InitChannel := FALSE;

IF udiDataSize > 0 THEN
	IF pOutputData <> TC3_MEMMAN.NULL THEN
		m_uinDataSize := udiDataSize;
		m_pOutputData := pOutputData;
		m_eState := E_PlcSaberDHCState.Init;
		InitChannel := TRUE;
	END_IF
END_IF

                      
END_METHOD
END_FUNCTION_BLOCK

CONFIGURATION Application
  RESOURCE Base_Elements ON PLC
    VAR_GLOBAL CONSTANT  (* Global_Version - This function has been automatically generated from the project information. *)
      {attribute 'const_non_replaced'}
      stLibVersion_Base_Elements : ST_LibVersion := (iMajor := 0, iMinor := 0, iBuild := 1, iRevision := 66, sVersion := '0.0.1.66');
    END_VAR
    VAR_GLOBAL CONSTANT  (* ACL_Const *)
      cuinMaxConnections : UINT := 50;
    END_VAR
    VAR_GLOBAL CONSTANT  (* ADS_IndexGroup *)
      cGET_SYMHANDLE_BYNAME : UDINT := 16#F003;  (* "Index-Group/Offset", GET_SYMHANDLE_BYNAME *)
      cREAD_WRITE_SYMVAL_BYHANDLE : UDINT := 16#F005;  (* "Index-Group/Offset", READ_WRITE_SYMVAL_BYHANDLE *)
    END_VAR
    VAR_GLOBAL CONSTANT  (* BCD_CmdState *)
      cBCD_CMD_DONE : INT := -1;  (* ctrl commands definitions *)
      cBCD_CMD_CONNECT_SOCKET : INT := 1002;  (* Connect TCP socket *)
      cBCD_CMD_CLOSE_SOCKET : INT := 1004;  (* Close TCP socket *)
      cBCD_CMD_COM_TEST : INT := 1006;  (* Communication test *)
      cBCD_CMD_READ_DEV_INFO : INT := 1008;  (* Readout device information *)
      cBCD_CMD_READ_OP_DATA : INT := 1010;  (* Readout operating data *)
      cBCD_CMD_READ_SERVICE_INFO : INT := 1012;  (* Readout service information *)
      cBCD_CMD_READ_BARCODE : INT := 1014;  (* Command enable the sensor gate for X-TIME ("duration" setting of sensor object trigger) *)
      cBCD_STA_WaitForJob : INT := 1000;  (* Sensor try to detect a barcode. ctrl state definitions *)
      cBCD_STA_ConnectSocketBusy : INT := 1002;  (* Open TCP socket busy *)
      cBCD_STA_CloseSocketBusy : INT := 1004;  (* Close TCP socket busy *)
      cBCD_STA_SocketClosed : INT := 1006;  (* TCP socket closed *)
      cBCD_STA_ComTestBusy : INT := 1008;  (* Communication test busy *)
      cBCD_STA_ReadCodeBusy : INT := 1010;  (* Read bar code busy *)
      cBCD_STA_Error : INT := 256;  (* Error *)
    END_VAR
    VAR_GLOBAL CONSTANT  (* PRS_CmdState *)
      cSTA_PRESENTBusy : INT := 201;  (* ctrl commands definitions specific commands >200 - every command has to be a even number ctrl specific states definitions *)
      cSTA_PRESENT : INT := 202;
      cSTA_ABSENTBusy : INT := 203;
      cSTA_ABSENT : INT := 204;
    END_VAR
    VAR_GLOBAL CONSTANT  (* RFD_Cmd *)
      cRFD_STA_Error : INT := 256;  (* ctrl state definitions Error *)
      cRFD_STA_PowerOnBusy : INT := 999;  (* Power On *)
      cRFD_STA_WaitForJob : INT := 1002;
      cRFD_STA_ResetBusy : INT := 1003;  (* RESET Reader *)
      cRFD_STA_OffBusy : INT := 1007;  (* Turn Off antenna *)
      cRFD_STA_Off : INT := 1008;
      cRFD_STA_WriteBusy : INT := 1009;  (* Write Data to Tag *)
      cRFD_STA_ReadBusy : INT := 1011;  (* Read Data from Tag *)
      cRFD_STA_TagInitBusy : INT := 1013;  (* Tag initialisation *)
      cRFD_STA_CheckBusy : INT := 1017;  (* Check connection to antenna *)
      cRFD_STA_MDSBusy : INT := 1019;  (* Service function read MDS-State (State of the near Tag) *)
      cRFD_STA_SLGBusy : INT := 1021;  (* Service function read SLG State (State of the antenna) *)
      cRFD_CMD_DONE : INT := -1;  (* ctrl commands definitions specific commands >200 - every command has to be a even number *)
      cRFD_CMD_CTRL_ON : INT := 1000;  (* Switch controller on *)
      cRFD_CMD_CTRL_OFF : INT := 1006;  (* Switch controller off *)
      cRFD_CMD_Write : INT := 1010;  (* Write Data to Tag *)
      cRFD_CMD_Read : INT := 1012;  (* Read Data from Tag *)
      cRFD_CMD_Check : INT := 1018;  (* Check connection to antenna *)
      cRFD_CMD_MDS : INT := 1020;  (* Service function read MDS-State (State of the near Tag) *)
      cRFD_CMD_SLG : INT := 1022;  (* Service function read SLG State (State of the antenna) *)
      cRFD_SUB_SetBaudrate : INT := 2001;  (* Sub States Power On Busy *)
      cRFD_SUB_SetComSettings : INT := 2002;  (* Set Communication Settings *)
      cRFD_SUB_ClearBuffer : INT := 2003;  (* Clear Buffer *)
      cRFD_SUB_InitString : INT := 2004;  (* Initialisation String sending *)
      cRFD_SUB_CheckPon : INT := 2005;  (* Check Power On State *)
      cRFD_SUB_Prepare : INT := 2010;  (* OFF Busy *)
      cRFD_SUB_SendBusy : INT := 2011;  (* Data send *)
      cRFD_SUB_WaitAnswer : INT := 2012;  (* Wait Answer *)
      cRFD_SUB_Write1 : INT := 2020;  (* SLG Write Mode 1 *)
      cRFD_SUB_Wait1 : INT := 2021;  (* SLG Wait Mode 1 *)
      cRFD_SUB_Write6 : INT := 2022;  (* SLG Write Mode 6 *)
      cRFD_SUB_Wait6 : INT := 2023;  (* SLG Wait Mode 6 *)
      cRFD_SUB_SubStatesEnd : INT := 2100;  (* Substates finished *)
    END_VAR
    VAR_GLOBAL CONSTANT  (* BCC_CmdState *)
      cBCC_CMD_READ : INT := 202;  (* ctrl commands definitions specific commands >200 - every command has to be a even number *)
      cBCC_STA_READBusy : INT := 201;  (* ctrl specific states definitions *)
      cBCC_STA_READ : INT := cBCC_CMD_READ;
      cSUB_READDELAYBusy : INT := 300;
      cSUB_SENDREADCOMMAND : INT := 301;
      cSUB_READBusy : INT := 302;
      cSUB_CLOSESOCKETstart : INT := 310;
      cSUB_CLOSESOCKETbusy : INT := 311;
      cSUB_CONNECTSOCKETstart : INT := 312;
      cSUB_CONNECTSOCKETbusy : INT := 313;
      cSUB_TESTSOCKETstart : INT := 314;
      cSUB_TESTSOCKETbusy : INT := 315;
      cSUB_DONE : INT := 316;
    END_VAR
    VAR_GLOBAL CONSTANT  (* CYL_CmdState *)
      cCMD_RETRACT : INT := 202;  (* ctrl commands definitions specific commands >200 - every command has to be a even number *)
      cCMD_EXTEND : INT := 204;
      cSTA_RETRACTBusy : INT := 201;  (* ctrl specific states definitions *)
      cSTA_RETRACT : INT := CYL_CmdState.cCMD_RETRACT;
      cSTA_EXTENDBusy : INT := 203;
      cSTA_EXTEND : INT := CYL_CmdState.cCMD_EXTEND;
    END_VAR
    VAR_GLOBAL CONSTANT  (* Const_DRV *)
      cMAX_BLOCKED_SUP : INT := 3;
    END_VAR
    VAR_GLOBAL CONSTANT  (* ECD_Const *)
      cuinMaxSlaves : UINT := 256;
    END_VAR
    VAR_GLOBAL CONSTANT  (* RFID_Data *)
      cRFID_RepetionID : DWORD := 16#10100;  (* RFID Data connection See RFID Specification Defines the Start Adress and the lengh of the Data in the RF ID Tag Every DoubleWord has to Words, Higher is lengh, lower word is Startadress Example 16#010005 => Startadress 5 Byte 1 => UV Settings *)
      cRFID_TrayInfo : DWORD := 16#10101;
      cRFID_HeighOfTray : DWORD := 16#10102;
      cRFID_Pretreatment : DWORD := 16#10103;
      cRFID_UVcuring : DWORD := 16#10104;
      cRFID_Filename : DWORD := 16#80105;
      cRFID_Brush : DWORD := 16#1010D;
      cRFID_TrayID : DWORD := 16#E0000;
      cRFID_TagID : DWORD := 16#8FFF0;
      cRFID_AllData : DWORD := 16#F0100;
    END_VAR
    VAR_GLOBAL CONSTANT  (* RFW_CmdState *)
      cCMD_ON : INT := 202;  (* ctrl commands definitions specific commands >200 - every command has to be a even number *)
      cCMD_READ : INT := 204;
      cCMD_WRITE : INT := 206;
      cSTA_ONBusy : INT := 201;  (* ctrl specific states definitions *)
      cSTA_ON : INT := cCMD_ON;
      cSTA_READBusy : INT := 203;
      cSTA_READ : INT := cCMD_READ;
      cSTA_WRITEBusy : INT := 205;
      cSTA_WRITE : INT := cCMD_WRITE;
    END_VAR
    VAR_GLOBAL CONSTANT  (* UMC_CmdState *)
      cCMD_RIGHT : INT := 202;  (* ctrl commands definitions specific commands >200 - every command has to be a even number *)
      cCMD_LEFT : INT := 204;
      cSTA_RESETMOTORERROR : INT := 203;  (* ctrl specific states definitions *)
    END_VAR
    VAR_GLOBAL CONSTANT  (* VLV_CmdState *)
      cCMD_OPEN : INT := 202;  (* ctrl commands definitions specific commands >200 - every command has to be a even number *)
      cCMD_CLOSE : INT := 204;
      cSTA_OPENBusy : INT := 201;  (* ctrl specific states definitions *)
      cSTA_OPEN : INT := VLV_CmdState.cCMD_OPEN;
      cSTA_CLOSEBusy : INT := 203;
      cSTA_CLOSE : INT := VLV_CmdState.cCMD_CLOSE;
    END_VAR
    VAR_GLOBAL CONSTANT  (* VPC_CmdState *)
      cSTA_VPC_StabilizeBusy : INT := 201;  (* ctrl specific states definitions *)
    END_VAR
    VAR_GLOBAL CONSTANT  (* ItemConst *)
      MAX_OVEN_SEGMENTS : UINT := 7;
      MAX_PRINT_HEAD_COUNT : UINT := 5;
      MAX_PRINT_MODULE_COUNT : UINT := 2;
    END_VAR
    VAR_GLOBAL CONSTANT  (* IdBaseConst *)
      cRECVDATACHANNELBUFFER : INT := 20;
    END_VAR
  END_RESOURCE
END_CONFIGURATION
